// TIA Portal V15.1 export
// export: Created 2026-01-09T13:45:12.6414146Z, ExportSetting WithDefaults, WithReadOnly, DisplayName Totally Integrated Automation Portal, DisplayVersion V15.1 Update 8, DisplayName TIA Portal Openness, DisplayVersion V15.1 Update 8, DisplayName STEP 7 Professional, DisplayVersion V15.1 Update 8, DisplayName WinCC Advanced, DisplayVersion V15.1 Update 8
FUNCTION_BLOCK "10.TIMER_CLOCK"   // FB10, LAD
{ S7_Optimized_Access := 'TRUE' }
VERSION : 0.1
// stored: AutoNumber false, CodeModifiedDate 2025-08-27T17:13:37.9521369Z, CompileDate 2025-08-30T17:40:34.6172449Z, CreationDate 2024-10-12T12:36:08.0193576Z, DownloadWithoutReinit false, HandleErrorsWithinBlock false, InterfaceModifiedDate 2023-08-14T08:08:19.3737097Z, IsConsistent true, IsIECCheckEnabled false, IsKnowHowProtected false, IsRetainMemResEnabled false, IsWriteProtected false, LibraryConformanceStatus The object is library-conformant., MemoryReserve 100, ModifiedDate 2025-08-27T17:13:37.9521369Z, ParameterModified 2022-05-24T16:04:05.0982286Z, PLCSimAdvancedSupport false, SetENOAutomatically False, StructureModified 2023-08-14T08:08:19.3737097Z, UDAEnableTagReadback false
   VAR_INPUT
      ON : Bool;
      CLOCK_1S : Bool;
      T_ON : Real;
      T_OFF : Real;
   END_VAR
   VAR_OUTPUT
      OUT : Bool;
   END_VAR
   VAR RETAIN
      TON : Real;
      TOFF : Real;
   END_VAR
   VAR
      CLK1 : Bool;
   END_VAR
   VAR_TEMP   // added for the SCL form of the ladder/FBD networks
      _w1 : Bool;
   END_VAR
BEGIN

REGION Network 1
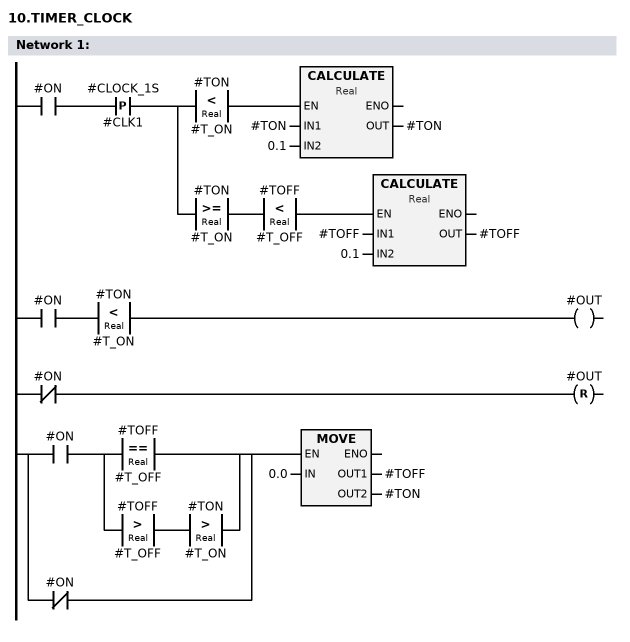
   RUNG wire#powerrail
      Contact( #ON )
      P_Contact(operand := #CLOCK_1S, bit := #CLK1)
      wire#w1
      { S7_Templates := "SrcType := Real" } LT_Contact(in1 := #TON, in2 := #T_ON)
      { S7_Templates := "SrcType := Real"; S7_Expression := "IN1+IN2" } Calculate(in1 := #TON, in2 := 0.1, out => #TON)
   END_RUNG
   RUNG wire#w1
      { S7_Templates := "SrcType := Real" } GE_Contact(in1 := #TON, in2 := #T_ON)
      { S7_Templates := "SrcType := Real" } LT_Contact(in1 := #TOFF, in2 := #T_OFF)
      { S7_Templates := "SrcType := Real"; S7_Expression := "IN1+IN2" } Calculate(in1 := #TOFF, in2 := 0.1, out => #TOFF)
   END_RUNG
   RUNG wire#powerrail
      Contact( #ON )
      { S7_Templates := "SrcType := Real" } LT_Contact(in1 := #TON, in2 := #T_ON)
      Coil( #OUT )
   END_RUNG
   RUNG wire#powerrail
      I_Contact( #ON )
      R_Coil( #OUT )
   END_RUNG
   RUNG wire#powerrail
      Contact( #ON )
      wire#w2
      { S7_Templates := "SrcType := Real" } EQ_Contact(in1 := #TOFF, in2 := #T_OFF)
      wire#w3
      Move(in := 0.0, out1 => #TOFF, out2 => #TON)
   END_RUNG
   RUNG wire#w2
      { S7_Templates := "SrcType := Real" } GT_Contact(in1 := #TOFF, in2 := #T_OFF)
      { S7_Templates := "SrcType := Real" } GT_Contact(in1 := #TON, in2 := #T_ON)
   END_RUNG wire#w3
   RUNG wire#powerrail
      I_Contact( #ON )
   END_RUNG wire#w3
   // the same network as SCL:
   #_w1 := #ON AND #CLOCK_1S AND NOT #CLK1;   // rising edge of #CLOCK_1S
   #CLK1 := #CLOCK_1S;
   IF #_w1 AND (#TON < #T_ON) THEN #TON := #TON+0.1; END_IF;
   IF #_w1 AND (#TON >= #T_ON) AND (#TOFF < #T_OFF) THEN #TOFF := #TOFF+0.1; END_IF;
   #OUT := #ON AND (#TON < #T_ON);
   IF NOT #ON THEN #OUT := FALSE; END_IF;
   IF (#ON AND ((#TOFF = #T_OFF) OR ((#TOFF > #T_OFF) AND (#TON > #T_ON)))) OR NOT #ON THEN
       #TOFF := 0.0;
       #TON := 0.0;
   END_IF;
END_REGION
END_FUNCTION_BLOCK
